FUNCTION_BLOCK TwoConCtlMulticast (* Composite Function Block Type for Multicast *)
  (* Standard: 61499-2 *)
  (* Version 0.2, 2003-12-05, JHC, Rockwell Automation, Renamed from NEWCOMPFB. *)
  (* Version 0.1, 2002-01-08, JHC, Rockwell Automation, Added DLY FB as example. *)
  (* Version 0.0, 2000-05-27, JHC, Rockwell Automation *)
  (* Compiler header: package fb.rt.cs725; *)
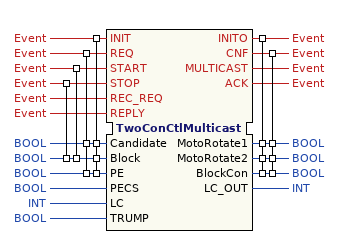
  EVENT_INPUT
    INIT WITH Candidate, Block, PE; (* Initialization Request *)
    REQ WITH Candidate, PE; (* Normal Execution Request *)
    START WITH Block;
    STOP WITH Block;
    REC_REQ;
    REPLY;
  END_EVENT
  EVENT_OUTPUT
    INITO WITH MotoRotate1, MotoRotate2, BlockCon; (* Initialization Confirm *)
    CNF WITH MotoRotate1, MotoRotate2, BlockCon; (* Execution Confirmation *)
    MULTICAST;
    ACK;
  END_EVENT
  VAR_INPUT
    Candidate : BOOL;
    Block : BOOL;
    PE : BOOL;
    PECS : BOOL;
    LC : INT;
    TRUMP : BOOL;
  END_VAR
  VAR_OUTPUT
    MotoRotate1 : BOOL;
    MotoRotate2 : BOOL;
    BlockCon : BOOL;
    LC_OUT : INT;
  END_VAR
  FBS
    FC11 : ConveyorCTL(PE := 0, Block := 0, Candidate := 0);
    FC12Multicast : ConveyorCTLMulticast;
  END_FBS
  EVENT_CONNECTIONS
    INIT TO FC11.INIT;
    REQ TO FC11.REQ;
    FC11.INITO TO FC12Multicast.INIT;
    FC12Multicast.START TO FC11.CAS_START;
    FC12Multicast.STOP TO FC11.CAS_STOP;
    REQ TO FC12Multicast.REQ;
    FC12Multicast.ACK TO ACK;
    FC12Multicast.MULTICAST TO MULTICAST;
    REC_REQ TO FC12Multicast.REC_REQ;
    REPLY TO FC12Multicast.REPLY;
  END_CONNECTIONS
  DATA_CONNECTIONS
    FC11.MotoRotate TO MotoRotate1;
    PE TO FC12Multicast.PE;
    Block TO FC12Multicast.Block;
    Candidate TO FC12Multicast.Candidate;
    FC12Multicast.MotoRotate TO MotoRotate2;
    FC12Multicast.BlockCon TO BlockCon;
    PECS TO FC12Multicast.PECS;
    LC TO FC12Multicast.LC;
    TRUMP TO FC12Multicast.TRUMP;
    FC12Multicast.LC_OUT TO LC_OUT;
  END_CONNECTIONS
END_FUNCTION_BLOCK
